// TwinCAT 3 PLC project IntegrationProjectsTests
// Title: IntegrationProjectsTests
// Company: Vortex.Library
// ProjectVersion: 0.4.2.535
// ProgramVersion: 3.1.4024.12
// libraries:
//   IntegrationProjects, 0.4.2.535 (Vortex.Library)
//   Tc2_Standard, * (Beckhoff Automation GmbH)
//   Tc2_System, * (Beckhoff Automation GmbH)
//   Tc3_Module, * (Beckhoff Automation GmbH)
//   TcoCore, 0.4.2.535 (Vortex.Library)
//   TcoData, 0.4.2.535 (Vortex.Library)
//   TcoDrivesBeckhoff, 0.4.2.535 (Vortex.Library)
//   TcoElements, 0.4.2.535 (Vortex.Library)
//   TcoIoBeckhoff, 0.4.2.535 (Vortex.Library)
//   TcoPneumatics, 0.4.2.535 (Vortex.Library)
// project tree:
//   / PlcTask.TcTTO
//   POUs/ MAIN.TcPOU, SampleComponentTests.TcPOU

CONFIGURATION IntegrationProjectsTests
    RESOURCE PLC ON TwinCAT3
        TASK PlcTask(INTERVAL := T#10ms, PRIORITY := 21);
        PROGRAM MAIN WITH PlcTask : MAIN;
    END_RESOURCE
END_CONFIGURATION

// ---- POUs/MAIN.TcPOU
PROGRAM MAIN
VAR
	_sampleComponentTests : SampleComponentTests;
END_VAR

END_PROGRAM

// ---- POUs/SampleComponentTests.TcPOU
FUNCTION_BLOCK SampleComponentTests EXTENDS _internals_TcoContext
VAR
	_sut : IntegrationProjects.SampleComponent(THIS^);
END_VAR

{attribute 'TcRpcEnable'}
METHOD INTERNAL AddTwoNumbersTest : INT
VAR_INPUT
	NumberOne : INT;
	NumberTwo : INT;
END_VAR
AddTwoNumbersTest := _sut.AddTwoNumbers(NumberOne, NumberTwo);
END_METHOD

METHOD PROTECTED Main
END_METHOD

{attribute 'TcRpcEnable'}
METHOD INTERNAL WaitForModuloTest : BOOL
VAR_INPUT
	Modulo : INT;
END_VAR
WaitForModuloTest := _sut.WaitForModulo(Modulo);
END_METHOD

END_FUNCTION_BLOCK
